// TIA Portal V18 export
DATA_BLOCK "LIVE_BLINK_MONITOR_DB"   // DB57
VERSION : 0.1
// stored: AutoNumber true, DBAccessibleFromOPCUA true, InstanceOfName LIVE_BLINK_MONITOR, InstanceOfType FB
"LIVE_BLINK_MONITOR"
   // VAR_INPUT
   //    high_in : Bool;
   //    flash_in : Bool;
   //    t_out : Time;
   //    t_resetER : Time;
   // END_VAR
   // VAR_OUTPUT
   //    ER_no_life : Bool;
   //    remTime : Time;
   // END_VAR
   // VAR
   //    tonS { S7_SetPoint := 'True'} : TON_TIME;
   //    was { S7_SetPoint := 'True'} : Bool;
   //    tonR { S7_SetPoint := 'True'} : TOF_TIME;
   //    flashing_ok : Bool;
   //    flashing_er : Bool;
   //    high_er : Bool;
   // END_VAR
BEGIN
END_DATA_BLOCK
